FUNCTION_BLOCK FB_PID_PWM
VAR_INPUT
	i_rSignal					:REAL;
	i_FreqMs					:REAL;
END_VAR
VAR_OUTPUT
	q_bPWM_Cmd					:BOOL;
END_VAR
VAR
	tonSignalOFF				:TON;
	tofSignalON					:TOF;
	Multiplier					:REAL;
END_VAR

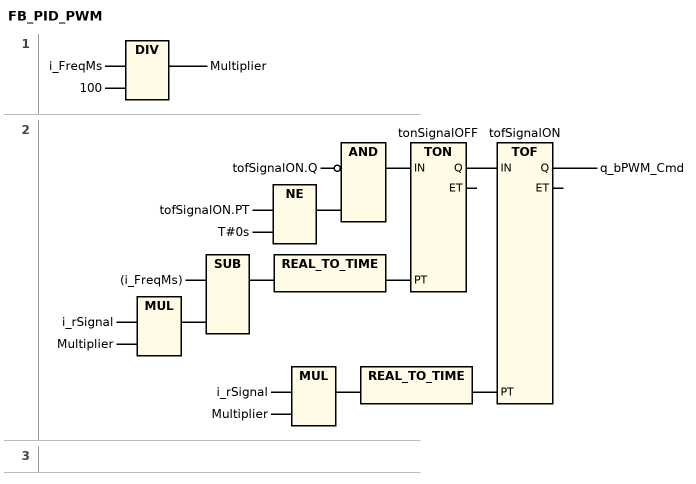
// NETWORK 1
Multiplier := i_FreqMs / 100;

// NETWORK 2
tonSignalOFF(IN := NOT tofSignalON.Q AND tofSignalON.PT <> T#0s, PT := REAL_TO_TIME(((i_FreqMs)) - i_rSignal * Multiplier)); // TON
tofSignalON(IN := tonSignalOFF.Q, PT := REAL_TO_TIME(i_rSignal * Multiplier)); // TOF
q_bPWM_Cmd := tofSignalON.Q;

// NETWORK 3

END_FUNCTION_BLOCK

(* stored: Version 1.1.0.1, ProductVersion 3.1.4024.12
   POU FB_PID_PWM: Id {6ff8a9bf-4654-420e-8c3b-084d521073ce}, SpecialFunc None *)
